INTERFACE I_RpcManager

METHOD PUBLIC TryHandleIncomingRequest : BOOL
VAR_INPUT
	Request : I_Request;
	Response : I_ServerResponse;
END_VAR
END_METHOD

END_INTERFACE

(* stored: Version 1.1.0.1, ProductVersion 3.1.4024.12
   Itf I_RpcManager: Id {a54b94bc-eef2-03ad-1a5d-2934e53ab2a3}
   Method TryHandleIncomingRequest: Id {89046c5d-d5ed-0b8b-00f2-6bbc260773b0} *)
